TYPE ST_CircleSettings :
STRUCT
	bWrite				:BOOL:=FALSE;
	uiXCenter			:UINT:=150;
	uiYCenter			:UINT:=150;
	uiRadius			:UINT:=50;
	lrStartDeg			:LREAL :=0;
	lrEndDeg			:LREAL :=370;
END_STRUCT
END_TYPE

(* stored: Version 1.1.0.1, ProductVersion 3.1.4026.11
   DUT ST_CircleSettings: Id {a5239e9c-7f97-4be1-a261-fe7118863d21} *)
